// TIA Portal V18 export
DATA_BLOCK "DataloggingDB"   // DB98
{ S7_Optimized_Access := 'FALSE' }
VERSION : 0.1
// stored: AutoNumber true, DBAccessibleFromOPCUA true, IsOnlyStoredInLoadMemory false, IsWriteProtectedInAS false
   VAR RETAIN
      Enable : Bool := false;
      "TXt/csv" : Bool := false;
      "Sdcard/pendrive" : Int := 0;
      "trigger SD card logging" : Bool := false;
      "trigger pendrive logging" : Bool := false;
      Data : Struct
         "Date" : DTL := DTL#1970-01-01-00:00:00;
         "Time" : Time_Of_Day := TOD#00:00:00;
         "Blade Number" : String := '';
         operator : Int := 0;
         "Batch A" : String[25] := '';
         "Batch B" : String[25] := '';
         IDVCA : String[25] := '';
         IDVCB : String[25] := '';
         "Pressure outlet A" : Real := 0.0;
         "Pressure outlet B" : Real := 0.0;
         "Ratio Control Size" : Real := 0.0;
         "Ratio A100:B" : Real := 0.0;
         "Ratio Min" : Real := 0.0;
         "Ratio Max" : Real := 0.0;
         CPK : Real := 0.0;
         "Event Number" : UDInt := 0;
         Function : String[25] := '';
         Error : UDInt := 0;
         "Temp.inlet Heater A" : Real := 0.0;
         "Temp.At mixing  Block A" : Real := 0.0;
         "Temp.At mixing Block B" : Real := 0.0;
         "Temp.At Resin outlet" : Real := 0.0;
      END_STRUCT;
      "Data string" : Struct
         "Pressure outlet A" : String[25] := '';
         "Pressure outlet B" : String[25] := '';
         "Ratio Control Size" : String[25] := '';
         "Ratio A100:B" : String[25] := '';
         "Ratio Min" : String[25] := '';
         "Ratio Max" : String[25] := '';
         CPK : String[25] := '';
         Function : String[25] := '';
         "Temp.inlet Heater A" : String[25] := '';
         "Temp.At mixing  Block A" : String[25] := '';
         "Temp.At mixing Block B" : String[25] := '';
         "Temp.At Resin outlet" : String[25] := '';
         "Total A flush" : String[25] := '';
         "Total B flush" : String[25] := '';
         "Total Size" : String[25] := '';
         "metering Size" : String[25] := '';
         "Shot Size A" : String[25] := '';
         "Shot Size B" : String[25] := '';
         "Total Size A" : String[25] := '';
         "Total Size B" : String[25] := '';
      END_STRUCT;
      Data_1 : Struct
         "Total A flush" : Real := 0.0;
         "Total B flush" : Real := 0.0;
         "Total Size" : Real := 0.0;
         "metering Size" : Real := 0.0;
         "Total size A" : Real := 0.0;
         "Total size B" : Real := 0.0;
         "MOULD NOMINAL PRESSURE" : Real := 0.0;
      END_STRUCT;
      "Copy Flush A qty" : Bool := false;
      "Copy Dearate A Qty" : Bool := false;
      "Copy Flush B qty" : Bool := false;
      "Copy Dearate B Qty" : Bool := false;
      "Copy Ab Qty" : Bool := false;
      "Total Size calculation" : Struct
         "Previous value" : Real := 0.0;
         "volume dispensed" : Real := 0.0;
         "present value" : Real := 0.0;
         "Value to add" : Real := 0.0;
         "start copy" : Bool := false;
         "dosing running" : Bool := false;
      END_STRUCT;
      "Total Size A calculation" : Struct
         "Previous value" : Real := 0.0;
         "volume dispensed" : Real := 0.0;
         "present value" : Real := 0.0;
         "Value to add" : Real := 0.0;
         "start copy" : Bool := false;
         "dosing running" : Bool := false;
      END_STRUCT;
      "Total Size B calculation" : Struct
         "Previous value" : Real := 0.0;
         "volume dispensed" : Real := 0.0;
         "present value" : Real := 0.0;
         "Value to add" : Real := 0.0;
         "start copy" : Bool := false;
         "dosing running" : Bool := false;
      END_STRUCT;
      "Ready to Log" : Bool := false;
      "Log Done" : Bool := false;
      "No.of counts to calculate CPK" : Int := 0;
      "reset A flush" : Bool := false;
      "reset B flush" : Bool := false;
      "reset total Size" : Bool := false;
      "Process Data Start/Stop" : Real := 0.0;
      "30sec timer done" : Bool := false;
      datacollection : Struct
         day : String[4] := '';
         month : String[4] := '';
         year : String[6] := '';
         filename : String[15] := 'Dopag_';
      END_STRUCT;
      date_time : DTL;
      current_day : UDInt;
      previous_day : UDInt;
      current_week : UDInt;
      previous_week : UDInt;
      current_month : UDInt;
      previous_month : UDInt;
      day_changed : Bool;
      week_changed : Bool;
      month_changed : Bool;
      totalsizepreviousday : Real;
      totalsizeday : Real;
      totalsizeweek : Real;
      totalsizepreviousweek : Real;
      totalsizemonth : Real;
      totalsizepreviousmonth : Real;
      Total_Production_metering : Real;
      Total_Production_Prerun : Real;
      Total_Production_Ratiocheck : Real;
      Total_Production_regeneration : Real;
      Total_Production_Flush : Real;
      Total_Volume : Real;
      Reset_total_volume : Bool;
      "Metering%" : Real;
      "Prerun%" : Real;
      "Ratiocheck%" : Real;
      "Regen%" : Real;
      "Flush%" : Real;
      "Last reset" : DTL;
   END_VAR
BEGIN
END_DATA_BLOCK
